// TIA Portal project "SCDW_风机控制" (V17)

(* hardware
DEVICE "PLC_1"  S7-1200 Station
   slot 0: "Rack_0"  S7-1200 Rack  Rack  V1.0
   slot 1: "PLC_1"  CPU 1214C AC/DC/Rly  6ES7 214-1BG40-0XB0  V4.5
   slot 2: "DI_DQ_Module_1"  6ES7 223-1PL30-0XB0  V1.0
   slot 3: "DI_DQ_Module_2"  6ES7 223-1PL30-0XB0  V1.0
   slot 4: "DI_DQ_Module_3"  6ES7 223-1PL30-0XB0  V1.0
   slot 101: "CM_1241"  6ES7 241-1CH32-0XB0  V2.1
*)

// ===== PLC "PLC_1"  CPU 1214C AC/DC/Rly =====

VAR_GLOBAL   // PLC tag table "数字输入量模块3"
   "消音复位" AT %I6.2 : Bool;
   "燃气低压" AT %I6.3 : Bool;
   "燃气高压" AT %I6.4 : Bool;
   "燃气泄漏" AT %I6.5 : Bool;
   "急停" AT %I6.6 : Bool;
   "15#小火" AT %Q6.0 : Bool;
   "15#复位" AT %Q6.1 : Bool;
   "15#大火" AT %Q6.2 : Bool;
   "烧嘴电源" AT %Q6.5 : Bool;
   "蜂鸣器" AT %Q6.6 : Bool;
END_VAR

VAR_GLOBAL   // PLC tag table "数字输入量模块2"
   "11#小火反馈" AT %I4.0 : Bool;
   "11#故障反馈" AT %I4.1 : Bool;
   "11#大火反馈" AT %I4.2 : Bool;
   "12#小火反馈" AT %I4.3 : Bool;
   "12#故障反馈" AT %I4.4 : Bool;
   "12#大火反馈" AT %I4.5 : Bool;
   "13#小火反馈" AT %I4.6 : Bool;
   "13#故障反馈" AT %I4.7 : Bool;
   "13#大火反馈" AT %I5.0 : Bool;
   "14#小火反馈" AT %I5.1 : Bool;
   "14#故障反馈" AT %I5.2 : Bool;
   "14#大火反馈" AT %I5.3 : Bool;
   "15#小火反馈" AT %I5.4 : Bool;
   "15#故障反馈" AT %I5.5 : Bool;
   "15#大火反馈" AT %I5.6 : Bool;
   "9#大火" AT %Q4.0 : Bool;
   "10#小火" AT %Q4.1 : Bool;
   "10#复位" AT %Q4.2 : Bool;
   "10#大火" AT %Q4.3 : Bool;
   "11#小火" AT %Q4.4 : Bool;
   "11#复位" AT %Q4.5 : Bool;
   "11#大火" AT %Q4.6 : Bool;
   "12#小火" AT %Q4.7 : Bool;
   "12#复位" AT %Q5.0 : Bool;
   "12#大火" AT %Q5.1 : Bool;
   "13#小火" AT %Q5.2 : Bool;
   "13#复位" AT %Q5.3 : Bool;
   "13#大火" AT %Q5.4 : Bool;
   "14#小火" AT %Q5.5 : Bool;
   "14#复位" AT %Q5.6 : Bool;
   "14#大火" AT %Q5.7 : Bool;
END_VAR

VAR_GLOBAL   // PLC tag table "数字输入量模块1"
   "5#大火反馈" AT %I2.0 : Bool;
   "6#小火反馈" AT %I2.1 : Bool;
   "6#故障反馈" AT %I2.2 : Bool;
   "6#大火反馈" AT %I2.3 : Bool;
   "7#小火反馈" AT %I2.4 : Bool;
   "7#故障反馈" AT %I2.5 : Bool;
   "7#大火反馈" AT %I2.6 : Bool;
   "8#小火反馈" AT %I2.7 : Bool;
   "8#故障反馈" AT %I3.0 : Bool;
   "8#大火反馈" AT %I3.1 : Bool;
   "9#小火反馈" AT %I3.2 : Bool;
   "9#故障反馈" AT %I3.3 : Bool;
   "9#大火反馈" AT %I3.4 : Bool;
   "10#小火反馈" AT %I3.5 : Bool;
   "10#故障反馈" AT %I3.6 : Bool;
   "10#大火反馈" AT %I3.7 : Bool;
   "4#复位" AT %Q2.0 : Bool;
   "4#大火" AT %Q2.1 : Bool;
   "5#小火" AT %Q2.2 : Bool;
   "5#复位" AT %Q2.3 : Bool;
   "5#大火" AT %Q2.4 : Bool;
   "6#小火" AT %Q2.5 : Bool;
   "6#复位" AT %Q2.6 : Bool;
   "6#大火" AT %Q2.7 : Bool;
   "7#小火" AT %Q3.0 : Bool;
   "7#复位" AT %Q3.1 : Bool;
   "7#大火" AT %Q3.2 : Bool;
   "8#小火" AT %Q3.3 : Bool;
   "8#复位" AT %Q3.4 : Bool;
   "8#大火" AT %Q3.5 : Bool;
   "9#小火" AT %Q3.6 : Bool;
   "9#复位" AT %Q3.7 : Bool;
END_VAR

VAR_GLOBAL   // PLC tag table "cpu点表"
   "1#小火反馈" AT %I0.0 : Bool;
   "1#故障反馈" AT %I0.1 : Bool;
   "1#大火反馈" AT %I0.2 : Bool;
   "2#小火反馈" AT %I0.3 : Bool;
   "2#故障反馈" AT %I0.4 : Bool;
   "2#大火反馈" AT %I0.5 : Bool;
   "3#小火反馈" AT %I0.6 : Bool;
   "3#故障反馈" AT %I0.7 : Bool;
   "3#大火反馈" AT %I1.0 : Bool;
   "4#小火反馈" AT %I1.1 : Bool;
   "4#故障反馈" AT %I1.2 : Bool;
   "4#大火反馈" AT %I1.3 : Bool;
   "5#小火反馈" AT %I1.4 : Bool;
   "5#故障反馈" AT %I1.5 : Bool;
   "1#小火" AT %Q0.0 : Bool;
   "1#复位" AT %Q0.1 : Bool;
   "1#大火" AT %Q0.2 : Bool;
   "2#小火" AT %Q0.3 : Bool;
   "2#复位" AT %Q0.4 : Bool;
   "2#大火" AT %Q0.5 : Bool;
   "3#小火" AT %Q0.6 : Bool;
   "3#复位" AT %Q0.7 : Bool;
   "3#大火" AT %Q1.0 : Bool;
   "4#小火" AT %Q1.1 : Bool;
   "风压" AT %IW64 : Int;
END_VAR

FUNCTION "风机输出功能" : Void   // FC1, SCL
{ S7_Optimized_Access := 'FALSE' }
VERSION : 0.1
BEGIN
       // Network 1: 风机运行条件
       IF "风机输出功能".风机运行按钮 AND NOT "风机输出功能".风机故障反馈 THEN
           "风机输出功能".风机运行标志 := TRUE;
       ELSE
           "风机输出功能".风机运行标志 := FALSE;
       END_IF;

       // Network 2: 手动模式 - 手动频率*2
       IF "风机输出功能".风机运行标志 AND "风机输出功能".风机手动 THEN
           "风机输出功能".风机控制输出 := "风机输出功能".风机手动频率 * 2.0;
       END_IF;

       // Network 3: 自动模式
       IF "风机输出功能".风机运行标志 AND NOT "风机输出功能".风机手动 THEN
           "风机输出功能".风机控制输出 := "风机输出功能".风机自动输出;
       END_IF;

       // Network 4: 停止清零控制输出
       IF NOT "风机输出功能".风机运行按钮 THEN
           "风机输出功能".风机控制输出 := 0.0;
       END_IF;

       // Network 5: 停止清零变频器参数
       IF NOT "风机输出功能".风机运行按钮 THEN
           "风机输出功能".变频器通讯设定频率 := 0;
           "风机输出功能".变频器通讯设定运行 := 0;
       END_IF;

       // Network 6: 频率换算
       IF "风机输出功能".风机运行标志 THEN
           "风机输出功能".风机控制输出码值 := "风机输出功能".风机控制输出 / 2.0;
           "风机输出功能".风机反馈频率 := "风机输出功能".风机控制输出码值 * 100.0;
           "风机输出功能".变频器通讯设定频率 := REAL_TO_INT("风机输出功能".风机反馈频率);
       END_IF;

       // Network 7: 运行状态
       IF "风机输出功能".变频器通讯运行状态 > 0 THEN
           "风机输出功能".风机运行反馈 := TRUE;
       END_IF;
       IF "风机输出功能".变频器通讯运行状态 = 0 THEN
           "风机输出功能".风机运行反馈 := FALSE;
       END_IF;

       // Network 8: 故障状态
       IF "风机输出功能".变频器通讯运行状态 < 0 THEN
           "风机输出功能".风机故障反馈 := TRUE;
       END_IF;

       // Network 9: 复位标志故障恢复
       IF "风机输出功能".风机故障反馈 AND "风机输出功能".风机复位标志 AND "风机输出功能".变频器通讯运行状态 >= 0 THEN
           "风机输出功能".风机故障反馈 := FALSE;
       END_IF;

       // Network 10: 运行指令
       IF "风机输出功能".风机运行标志 THEN
           "风机输出功能".变频器通讯设定运行 := 1;
       END_IF;
END_FUNCTION

ORGANIZATION_BLOCK "Main"   // OB1, LAD, ProgramCycle
TITLE = "Main Program Sweep (Cycle)"
{ S7_Optimized_Access := 'TRUE' }
VERSION : 0.1
   VAR_INPUT
      Initial_Call : Bool;   // Initial call of this OB
      Remanence : Bool;   // =True, if remanent data are available
   END_VAR
BEGIN
END_ORGANIZATION_BLOCK